// TIA Portal V18 export
FUNCTION_BLOCK "_ML2_mode"   // FB45, FBD
{ S7_Optimized_Access := 'TRUE' }
VERSION : 0.1
// stored: AutoNumber true, IsIECCheckEnabled false, IsRetainMemResEnabled false, MemoryReserve 100, SetENOAutomatically false, UDAEnableTagReadback false
   VAR_IN_OUT
      xSoftSTOP : Bool;
      yExecuteAll : Bool;
      yTeam_unison : Bool;
      yOVERRIDE : Bool;
   END_VAR
BEGIN
END_FUNCTION_BLOCK
